{attribute addProperty BoxType "EK1100-0000-0018"}
{attribute addProperty Id "Beckhoff_ELM35xxEK1122Beckhoff_ELM35xxEK1122_B82F516C162A_0001_ELM3502_0000_0016ELM3502_1C598C2535244A_0002_ELM3502_0000_0017ELM3502_1C598C2535244A_0003_ELM3502_0000_0018ELM3502_1C598C2535244A_0004_ELM3502_0000_0019ELM3502_1C598C2535244A_0005_ELM3504_0000_0016ELM3504_EF18820948060A_0006_ELM3504_0000_0017ELM3504_EF18820948060A_0007_ELM3504_0000_0018ELM3504_EF18820948060A_0008_ELM3504_0000_0019ELM3504_EF18820948060"}
{attribute addProperty CRC "1963888361"}
{attribute addProperty SizeInBites "3344"}
{attribute addProperty SizeInBytes "418"}
TYPE Beckhoff_ELM35xx_750E8EE9 EXTENDS EK1100_179A0949 :
STRUCT
	{attribute addProperty Name "Beckhoff_ELM35xxEK1122"}
	Beckhoff_ELM35xxEK1122 : Beckhoff_ELM35xxEK1122_B82F516C;
	{attribute addProperty Name "A_0001_ELM3502_0000_0016"}
	A_0001_ELM3502_0000_0016 : ELM3502_1C598C25;
	{attribute addProperty Name "A_0002_ELM3502_0000_0017"}
	A_0002_ELM3502_0000_0017 : ELM3502_1C598C25;
	{attribute addProperty Name "A_0003_ELM3502_0000_0018"}
	A_0003_ELM3502_0000_0018 : ELM3502_1C598C25;
	{attribute addProperty Name "A_0004_ELM3502_0000_0019"}
	A_0004_ELM3502_0000_0019 : ELM3502_1C598C25;
	{attribute addProperty Name "A_0005_ELM3504_0000_0016"}
	A_0005_ELM3504_0000_0016 : ELM3504_EF188209;
	{attribute addProperty Name "A_0006_ELM3504_0000_0017"}
	A_0006_ELM3504_0000_0017 : ELM3504_EF188209;
	{attribute addProperty Name "A_0007_ELM3504_0000_0018"}
	A_0007_ELM3504_0000_0018 : ELM3504_EF188209;
	{attribute addProperty Name "A_0008_ELM3504_0000_0019"}
	A_0008_ELM3504_0000_0019 : ELM3504_EF188209;
END_STRUCT
END_TYPE

(* stored: Version 1.2.0.0, ProductVersion 3.1.4024.9
   DUT Beckhoff_ELM35xx_750E8EE9: Id {ce2c1479-e09b-4b67-9e5a-a91e728de953} *)
